// TIA Portal V18 export
FUNCTION_BLOCK "LED_Behavior"   // FB11, LAD
TITLE = Description:
{ S7_Optimized_Access := 'TRUE' }
VERSION : 0.1
// Old control block - should be checked and described.
// stored: AutoNumber true, IsIECCheckEnabled false, IsRetainMemResEnabled false, MemoryReserve 100, SetENOAutomatically false, UDAEnableTagReadback false
   VAR_INPUT
      RED : Bool;
      GREEN : Bool;
      RED_BLINK : Bool;
      GREEN_BLINK : Bool;
      RED_GREEN_BLINK : Bool;
   END_VAR
   VAR_OUTPUT
      LED_1_Output : Bool;
      LED_2_Output : Bool;
   END_VAR
   VAR
      Red_Blink_Output : Bool;
      Green_Blink_Output : Bool;
      "Red/Green_Blink_Output" : Bool;
      Red_Blink_M : Bool;
      Red_Blink_S : Bool;
      Green_Blink_M : Bool;
      Green_Blink_S : Bool;
      Reset_Red_Blink : Bool;
      Reset_Green_Blink : Bool;
      Reset_RED_GREEN_Blink : Bool;
      RG_Blink_M : Bool;
      RG_Blink_S : Bool;
   END_VAR
BEGIN

REGION Network 1: Output 1 Color 1=RED 0=GREEN
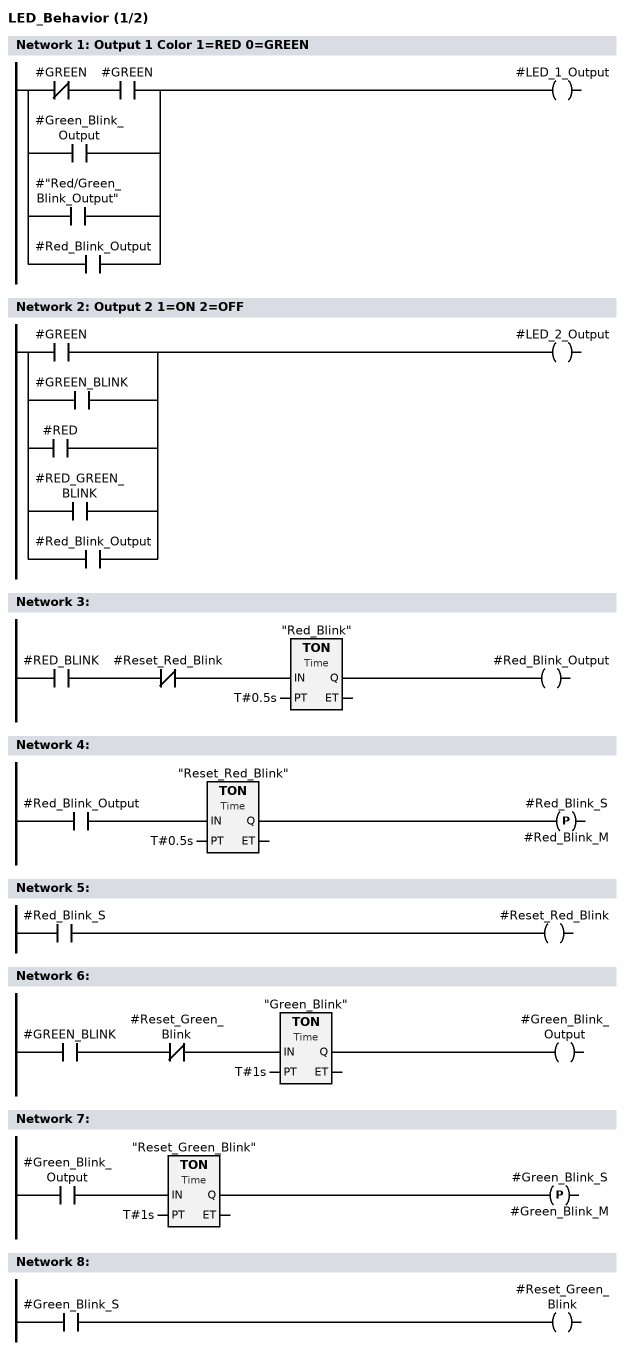
   RUNG wire#powerrail
      I_Contact( #GREEN )
      Contact( #GREEN )
      wire#w1
      Coil( #LED_1_Output )
   END_RUNG
   RUNG wire#powerrail
      Contact( #Green_Blink_Output )
   END_RUNG wire#w1
   RUNG wire#powerrail
      Contact( #"Red/Green_Blink_Output" )
   END_RUNG wire#w1
   RUNG wire#powerrail
      Contact( #Red_Blink_Output )
   END_RUNG wire#w1
   // the same network as SCL:
   #LED_1_Output := (NOT #GREEN AND #GREEN) OR #Green_Blink_Output OR #"Red/Green_Blink_Output" OR #Red_Blink_Output;
END_REGION

REGION Network 2: Output 2 1=ON 2=OFF
   RUNG wire#powerrail
      Contact( #GREEN )
      wire#w1
      Coil( #LED_2_Output )
   END_RUNG
   RUNG wire#powerrail
      Contact( #GREEN_BLINK )
   END_RUNG wire#w1
   RUNG wire#powerrail
      Contact( #RED )
   END_RUNG wire#w1
   RUNG wire#powerrail
      Contact( #RED_GREEN_BLINK )
   END_RUNG wire#w1
   RUNG wire#powerrail
      Contact( #Red_Blink_Output )
   END_RUNG wire#w1
   // the same network as SCL:
   #LED_2_Output := #GREEN OR #GREEN_BLINK OR #RED OR #RED_GREEN_BLINK OR #Red_Blink_Output;
END_REGION

REGION Network 3
   RUNG wire#powerrail
      Contact( #RED_BLINK )
      I_Contact( #Reset_Red_Blink )
      { S7_Templates := "time_type := Time" } "Red_Blink".TON(pt := T#0.5s, et =>)
      Coil( #Red_Blink_Output )
   END_RUNG
   // the same network as SCL:
   "Red_Blink".TON(IN := #RED_BLINK AND NOT #Reset_Red_Blink, PT := T#0.5s);
   #Red_Blink_Output := "Red_Blink".Q;
END_REGION

REGION Network 4
   "Reset_Red_Blink".TON(IN := #Red_Blink_Output, PT := T#0.5s);
   #Red_Blink_S := "Reset_Red_Blink".Q AND NOT #Red_Blink_M;   // rising edge
   #Red_Blink_M := "Reset_Red_Blink".Q;
END_REGION

REGION Network 5
   RUNG wire#powerrail
      Contact( #Red_Blink_S )
      Coil( #Reset_Red_Blink )
   END_RUNG
   // the same network as SCL:
   #Reset_Red_Blink := #Red_Blink_S;
END_REGION

REGION Network 6
   RUNG wire#powerrail
      Contact( #GREEN_BLINK )
      I_Contact( #Reset_Green_Blink )
      { S7_Templates := "time_type := Time" } "Green_Blink".TON(pt := T#1s, et =>)
      Coil( #Green_Blink_Output )
   END_RUNG
   // the same network as SCL:
   "Green_Blink".TON(IN := #GREEN_BLINK AND NOT #Reset_Green_Blink, PT := T#1s);
   #Green_Blink_Output := "Green_Blink".Q;
END_REGION

REGION Network 7
   "Reset_Green_Blink".TON(IN := #Green_Blink_Output, PT := T#1s);
   #Green_Blink_S := "Reset_Green_Blink".Q AND NOT #Green_Blink_M;   // rising edge
   #Green_Blink_M := "Reset_Green_Blink".Q;
END_REGION

REGION Network 8
   RUNG wire#powerrail
      Contact( #Green_Blink_S )
      Coil( #Reset_Green_Blink )
   END_RUNG
   // the same network as SCL:
   #Reset_Green_Blink := #Green_Blink_S;
END_REGION

REGION Network 9
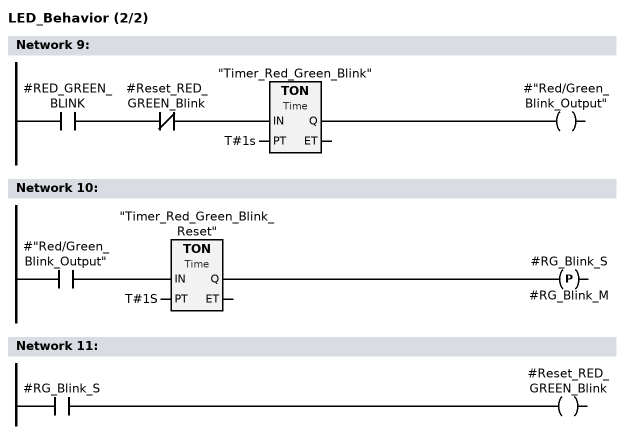
   RUNG wire#powerrail
      Contact( #RED_GREEN_BLINK )
      I_Contact( #Reset_RED_GREEN_Blink )
      { S7_Templates := "time_type := Time" } "Timer_Red_Green_Blink".TON(pt := T#1s, et =>)
      Coil( #"Red/Green_Blink_Output" )
   END_RUNG
   // the same network as SCL:
   "Timer_Red_Green_Blink".TON(IN := #RED_GREEN_BLINK AND NOT #Reset_RED_GREEN_Blink, PT := T#1s);
   #"Red/Green_Blink_Output" := "Timer_Red_Green_Blink".Q;
END_REGION

REGION Network 10
   "Timer_Red_Green_Blink_Reset".TON(IN := #"Red/Green_Blink_Output", PT := T#1S);
   #RG_Blink_S := "Timer_Red_Green_Blink_Reset".Q AND NOT #RG_Blink_M;   // rising edge
   #RG_Blink_M := "Timer_Red_Green_Blink_Reset".Q;
END_REGION

REGION Network 11
   RUNG wire#powerrail
      Contact( #RG_Blink_S )
      Coil( #Reset_RED_GREEN_Blink )
   END_RUNG
   // the same network as SCL:
   #Reset_RED_GREEN_Blink := #RG_Blink_S;
END_REGION
END_FUNCTION_BLOCK
